PROGRAM DatenRangieren
VAR	
	VersionsText: STRING := 'LAP 2010/5 Pumpensteuerung V2.0';
END_VAR

VersionsInfo.Ver := MAXSTRING_TO_BYTEARR(VersionsText);

SimDI.B1 := BitLesen(DigInput.DI[0],0);
SimDI.B2 := BitLesen(DigInput.DI[0],1);
SimDI.F1 := BitLesen(DigInput.DI[0],2);
SimDI.S1 := BitLesen(DigInput.DI[0],3);
SimDI.S2 := BitLesen(DigInput.DI[0],4);
SimDI.S3 := BitLesen(DigInput.DI[0],5);

DigOutput.DA[0] := AlleBitSetzen(	SimDa.P1,	
									SimDa.P2,	
									SimDa.Q1,
									FALSE, FALSE, FALSE, FALSE, FALSE);

END_PROGRAM

(* stored: Version 1.1.0.1, ProductVersion 3.1.4024.5
   POU DatenRangieren: Id {ad49a684-d9e6-4dba-bece-08745f191ac1}, SpecialFunc None *)
